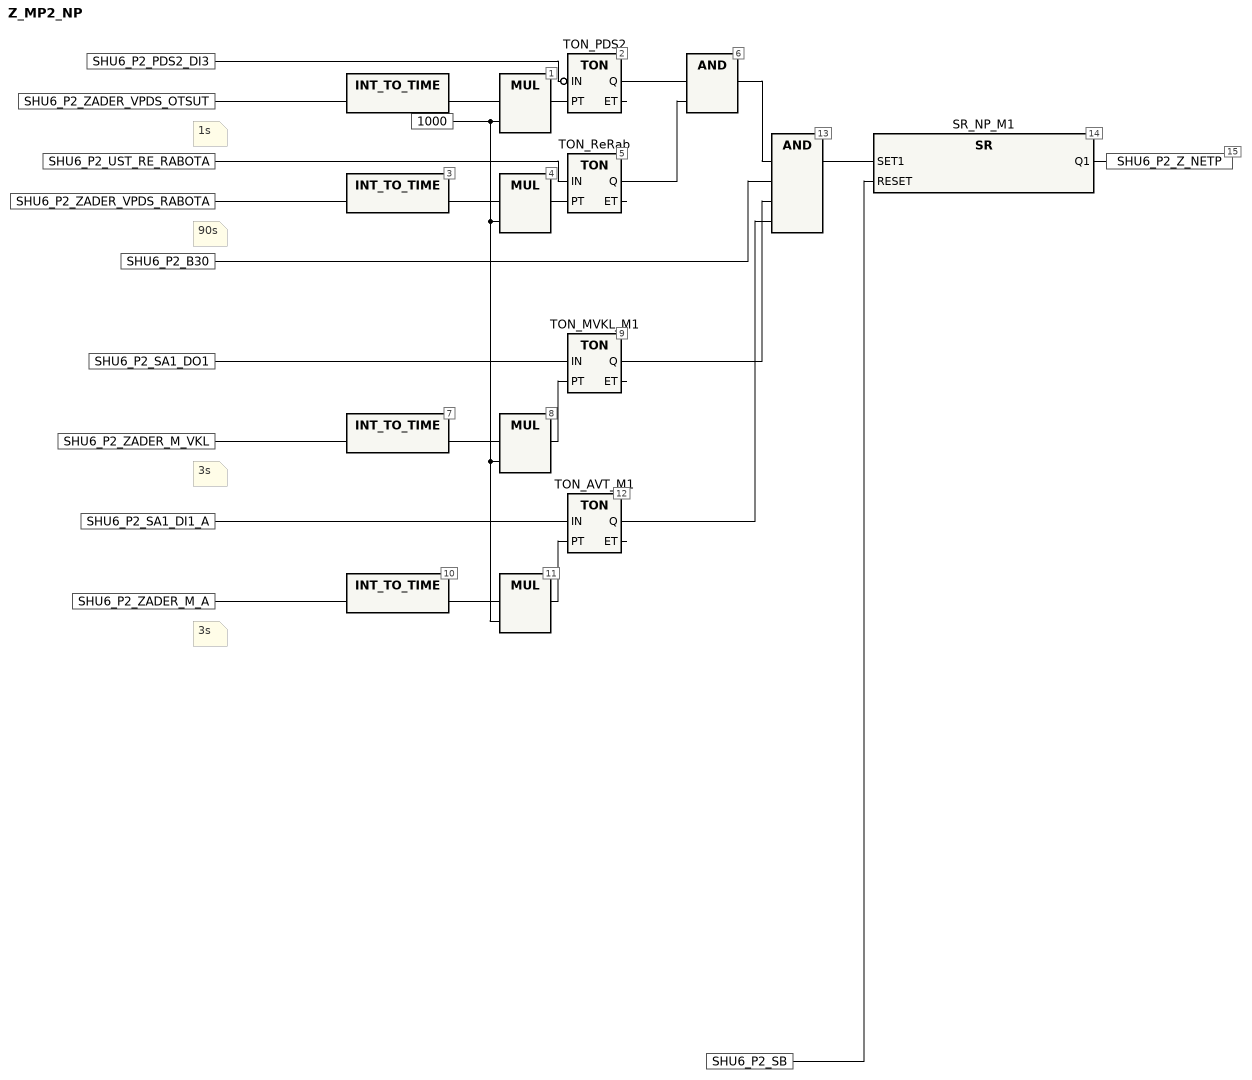
[picture p144: Z_MP2_NP (CFC)]
_CFC_ (* Continuous Function Chart, elements in execution order *)
(* 1s *)
(* 90s *)
(* 3s *)
(* 3s *)
#0 INT_TO_TIME(SHU6_P2_ZADER_VPDS_OTSUT)
#1 MUL(#0, 1000)
#2 TON_PDS2:TON(IN: NOT SHU6_P2_PDS2_DI3, PT: #1)
#3 INT_TO_TIME(SHU6_P2_ZADER_VPDS_RABOTA)
#4 MUL(#3, 1000)
#5 TON_ReRab:TON(IN: SHU6_P2_UST_RE_RABOTA, PT: #4)
#6 AND(#2.Q, #5.Q)
#7 INT_TO_TIME(SHU6_P2_ZADER_M_VKL)
#8 MUL(#7, 1000)
#9 TON_MVKL_M1:TON(IN: SHU6_P2_SA1_DO1, PT: #8)
#10 INT_TO_TIME(SHU6_P2_ZADER_M_A)
#11 MUL(#10, 1000)
#12 TON_AVT_M1:TON(IN: SHU6_P2_SA1_DI1_A, PT: #11)
#13 AND(#6, SHU6_P2_B30, #9.Q, #12.Q)
#14 SR_NP_M1:SR(SET1: #13, RESET: SHU6_P2_SB)
#15 SHU6_P2_Z_NETP <= #14.Q1
_END_CFC_
(* the same logic as Structured Text *)
(* 1s *)
(* 90s *)
(* 3s *)
(* 3s *)
TON_PDS2(IN := NOT SHU6_P2_PDS2_DI3, PT := INT_TO_TIME(SHU6_P2_ZADER_VPDS_OTSUT) * 1000);
TON_ReRab(IN := SHU6_P2_UST_RE_RABOTA, PT := INT_TO_TIME(SHU6_P2_ZADER_VPDS_RABOTA) * 1000);
TON_MVKL_M1(IN := SHU6_P2_SA1_DO1, PT := INT_TO_TIME(SHU6_P2_ZADER_M_VKL) * 1000);
TON_AVT_M1(IN := SHU6_P2_SA1_DI1_A, PT := INT_TO_TIME(SHU6_P2_ZADER_M_A) * 1000);
SR_NP_M1(SET1 := (TON_PDS2.Q AND TON_ReRab.Q) AND SHU6_P2_B30 AND TON_MVKL_M1.Q AND TON_AVT_M1.Q, RESET := SHU6_P2_SB);
SHU6_P2_Z_NETP := SR_NP_M1.Q1;
END_PROGRAM

(* POU TZBiS/TZB/Z_MV2/Z_MV2_NP, CFC *)
PROGRAM Z_MV2_NP
VAR
	TON_PDS2: TON;
	TON_ReRab: TON;
	TON_MVKL: TON;
	TON_AVT: TON;
	TP_SR: TP;
	SR_NP_M1: SR;
	SR_NP_M2: SR;
	TON_MVKL_M1: TON;
	TON_AVT_M1: TON;
	TON_AVT_M2: TON;
	TON_MVKL_M2: TON;
END_VAR
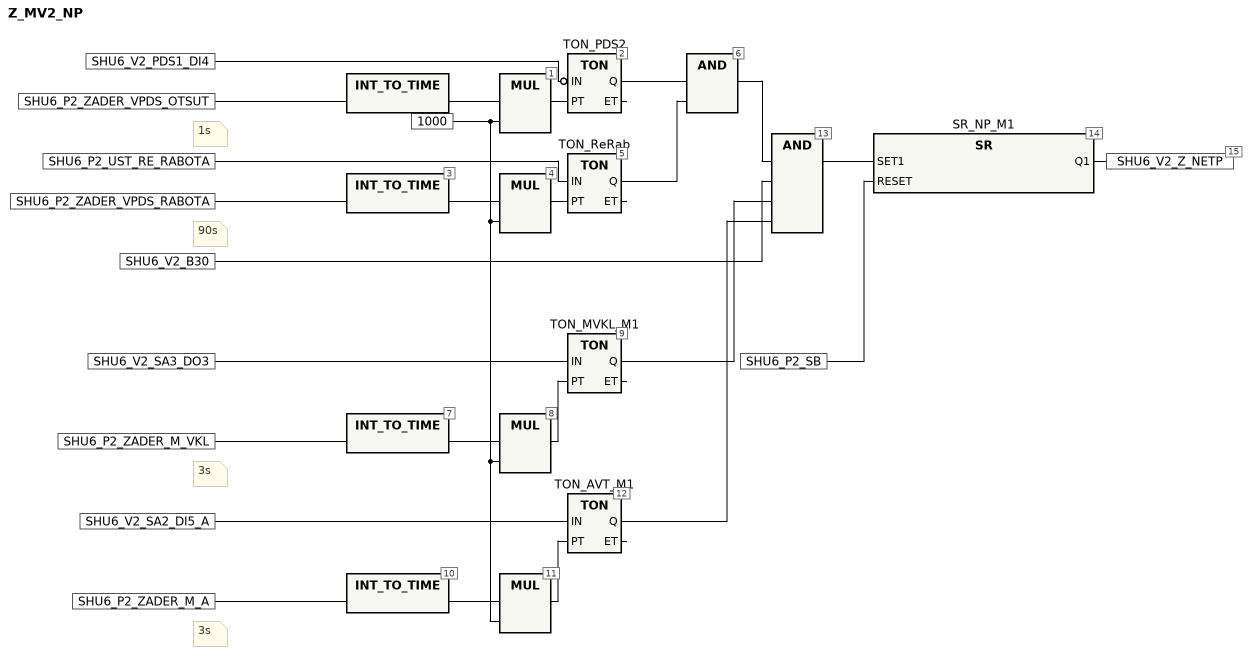
_CFC_ (* Continuous Function Chart, elements in execution order *)
(* 1s *)
(* 90s *)
(* 3s *)
(* 3s *)
#0 INT_TO_TIME(SHU6_P2_ZADER_VPDS_OTSUT)
#1 MUL(#0, 1000)
#2 TON_PDS2:TON(IN: NOT SHU6_V2_PDS1_DI4, PT: #1)
#3 INT_TO_TIME(SHU6_P2_ZADER_VPDS_RABOTA)
#4 MUL(#3, 1000)
#5 TON_ReRab:TON(IN: SHU6_P2_UST_RE_RABOTA, PT: #4)
#6 AND(#2.Q, #5.Q)
#7 INT_TO_TIME(SHU6_P2_ZADER_M_VKL)
#8 MUL(#7, 1000)
#9 TON_MVKL_M1:TON(IN: SHU6_V2_SA3_DO3, PT: #8)
#10 INT_TO_TIME(SHU6_P2_ZADER_M_A)
#11 MUL(#10, 1000)
#12 TON_AVT_M1:TON(IN: SHU6_V2_SA2_DI5_A, PT: #11)
#13 AND(#6, SHU6_V2_B30, #9.Q, #12.Q)
#14 SR_NP_M1:SR(SET1: #13, RESET: SHU6_P2_SB)
#15 SHU6_V2_Z_NETP <= #14.Q1
_END_CFC_
(* the same logic as Structured Text *)
(* 1s *)
(* 90s *)
(* 3s *)
(* 3s *)
TON_PDS2(IN := NOT SHU6_V2_PDS1_DI4, PT := INT_TO_TIME(SHU6_P2_ZADER_VPDS_OTSUT) * 1000);
TON_ReRab(IN := SHU6_P2_UST_RE_RABOTA, PT := INT_TO_TIME(SHU6_P2_ZADER_VPDS_RABOTA) * 1000);
TON_MVKL_M1(IN := SHU6_V2_SA3_DO3, PT := INT_TO_TIME(SHU6_P2_ZADER_M_VKL) * 1000);
TON_AVT_M1(IN := SHU6_V2_SA2_DI5_A, PT := INT_TO_TIME(SHU6_P2_ZADER_M_A) * 1000);
SR_NP_M1(SET1 := (TON_PDS2.Q AND TON_ReRab.Q) AND SHU6_V2_B30 AND TON_MVKL_M1.Q AND TON_AVT_M1.Q, RESET := SHU6_P2_SB);
SHU6_V2_Z_NETP := SR_NP_M1.Q1;
END_PROGRAM

(* POU TZBiS/TZB/Z_NET_VKH_NAPR, CFC *)
PROGRAM Z_NET_VKH_NAPR
VAR
	RS_Net_vhk_napr: SR;
	TON_KV: TON;
END_VAR
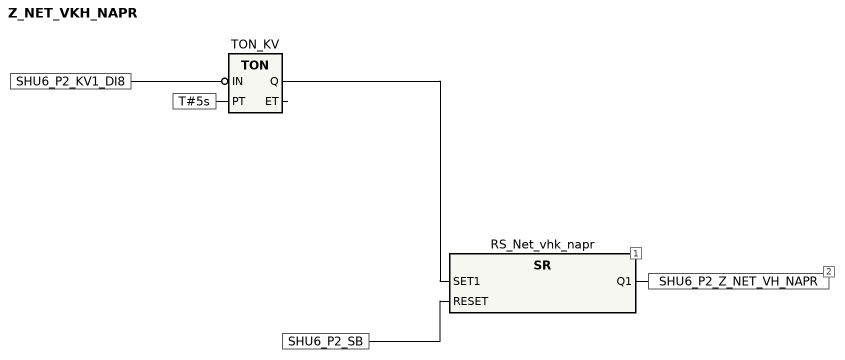
_CFC_ (* Continuous Function Chart, elements in execution order *)
#0 TON_KV:TON(IN: NOT SHU6_P2_KV1_DI8, PT: T#5s)
#1 RS_Net_vhk_napr:SR(SET1: #0.Q, RESET: SHU6_P2_SB)
#2 SHU6_P2_Z_NET_VH_NAPR <= #1.Q1
_END_CFC_
(* the same logic as Structured Text *)
TON_KV(IN := NOT SHU6_P2_KV1_DI8, PT := T#5s);
RS_Net_vhk_napr(SET1 := TON_KV.Q, RESET := SHU6_P2_SB);
SHU6_P2_Z_NET_VH_NAPR := RS_Net_vhk_napr.Q1;
END_PROGRAM

(* POU TZBiS/TZB/Z_OTKAZ_VTOR_ZEP, CFC *)
PROGRAM Z_OTKAZ_VTOR_ZEP
VAR
	rs_otkaz_vtor_sep: RS;
	TON_VTOR_ZEP: TON;
END_VAR
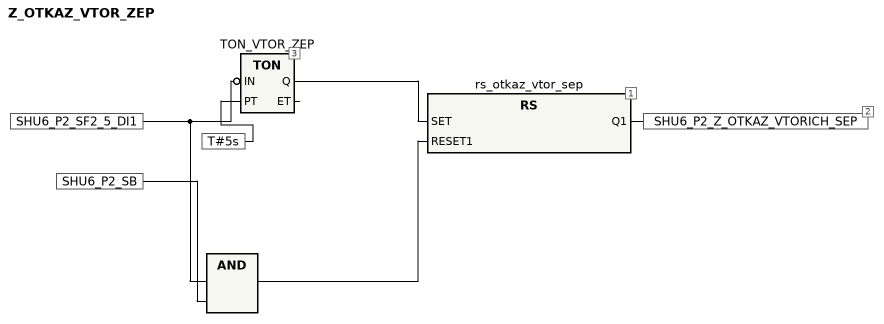
_CFC_ (* Continuous Function Chart, elements in execution order *)
#0 AND(SHU6_P2_SF2_5_DI1, SHU6_P2_SB)
#1 rs_otkaz_vtor_sep:RS(SET: #3.Q, RESET1: #0)
#2 SHU6_P2_Z_OTKAZ_VTORICH_SEP <= #1.Q1
#3 TON_VTOR_ZEP:TON(IN: NOT SHU6_P2_SF2_5_DI1, PT: T#5s)
_END_CFC_
(* the same logic as Structured Text *)
rs_otkaz_vtor_sep(SET := TON_VTOR_ZEP.Q, RESET1 := SHU6_P2_SF2_5_DI1 AND SHU6_P2_SB);
SHU6_P2_Z_OTKAZ_VTORICH_SEP := rs_otkaz_vtor_sep.Q1;
TON_VTOR_ZEP(IN := NOT SHU6_P2_SF2_5_DI1, PT := T#5s);
END_PROGRAM

(* POU TZBiS/TZB/Z_P1_NP, CFC *)
PROGRAM Z_P1_NP
VAR
	SR_P1_NPit: SR;
END_VAR
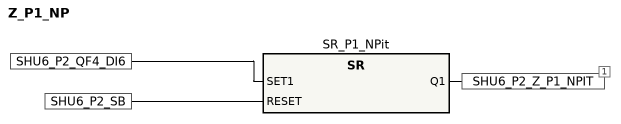
_CFC_ (* Continuous Function Chart, elements in execution order *)
#0 SR_P1_NPit:SR(SET1: SHU6_P2_QF4_DI6, RESET: SHU6_P2_SB)
#1 SHU6_P2_Z_P1_NPIT <= #0.Q1
_END_CFC_
(* the same logic as Structured Text *)
SR_P1_NPit(SET1 := SHU6_P2_QF4_DI6, RESET := SHU6_P2_SB);
SHU6_P2_Z_P1_NPIT := SR_P1_NPit.Q1;
END_PROGRAM

(* POU TZBiS/TZB/Sbros_All, CFC *)
PROGRAM Sbros_All
VAR
END_VAR
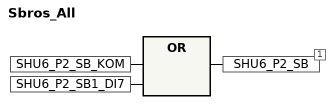
_CFC_ (* Continuous Function Chart, elements in execution order *)
#0 OR(SHU6_P2_SB_KOM, SHU6_P2_SB1_DI7)
#1 SHU6_P2_SB <= #0
_END_CFC_
(* the same logic as Structured Text *)
SHU6_P2_SB := SHU6_P2_SB_KOM OR SHU6_P2_SB1_DI7;
END_PROGRAM

(* POU TZBiS/TZB/Z_Pozhar, CFC *)
PROGRAM Z_Pozhar
VAR
	SR_Pozhar: SR;
END_VAR
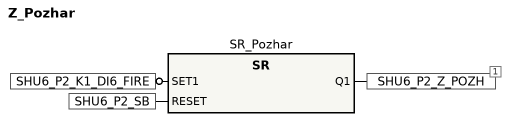
_CFC_ (* Continuous Function Chart, elements in execution order *)
#0 SR_Pozhar:SR(SET1: NOT SHU6_P2_K1_DI6_FIRE, RESET: SHU6_P2_SB)
#1 SHU6_P2_Z_POZH <= #0.Q1
_END_CFC_
(* the same logic as Structured Text *)
SR_Pozhar(SET1 := NOT SHU6_P2_K1_DI6_FIRE, RESET := SHU6_P2_SB);
SHU6_P2_Z_POZH := SR_Pozhar.Q1;
END_PROGRAM

(* POU TZBiS/TZB/Z_Zam, CFC *)
PROGRAM Z_Zam
VAR
	RT_VKL: R_TRIG;
	SR_ZAM: SR;
	TON_VKL: TON;
	TP_VKL: TON;
	FT_TP_VKL: F_TRIG;
	SR_TS: SR;
END_VAR
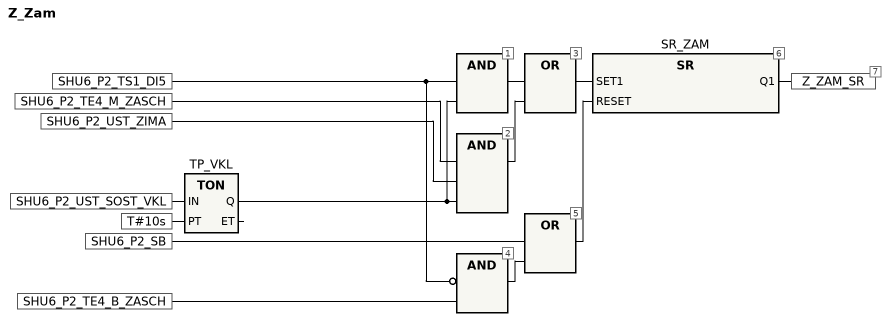
_CFC_ (* Continuous Function Chart, elements in execution order *)
#0 TP_VKL:TON(IN: SHU6_P2_UST_SOST_VKL, PT: T#10s)
#1 AND(SHU6_P2_TS1_DI5, #0.Q)
#2 AND(SHU6_P2_TE4_M_ZASCH, SHU6_P2_UST_ZIMA, #0.Q)
#3 OR(#1, #2)
#4 AND(NOT SHU6_P2_TS1_DI5, SHU6_P2_TE4_B_ZASCH)
#5 OR(SHU6_P2_SB, #4)
#6 SR_ZAM:SR(SET1: #3, RESET: #5)
#7 Z_ZAM_SR <= #6.Q1
_END_CFC_
(* the same logic as Structured Text *)
TP_VKL(IN := SHU6_P2_UST_SOST_VKL, PT := T#10s);
SR_ZAM(SET1 := (SHU6_P2_TS1_DI5 AND TP_VKL.Q) OR (SHU6_P2_TE4_M_ZASCH AND SHU6_P2_UST_ZIMA AND TP_VKL.Q), RESET := SHU6_P2_SB OR (NOT SHU6_P2_TS1_DI5 AND SHU6_P2_TE4_B_ZASCH));
Z_ZAM_SR := SR_ZAM.Q1;
END_PROGRAM

(* POU TZBiS/TZB/Z_Dlit_Ster_Reg, CFC *)
	PROGRAM Z_Dlit_Ster_Reg
VAR
	SR_HZ20S60: SR;
	LT_HZm20: ISTOK_LT;
	TON_HZm20: TON;
END_VAR
VAR (* helpers for the ST form of the networks *)
	_t19 : BOOL;
END_VAR
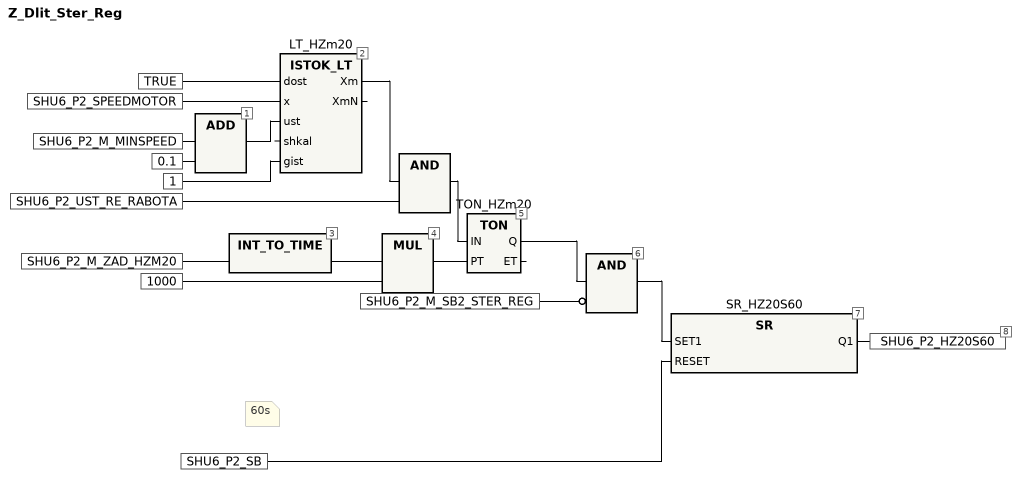
